Staubli VAL3: PlasticMain.pjx

--- PlasticMain.pjx ---
Parameters version=s7.0 stackSize=400000 millimeterUnit=true
Program file=__ts_english.pgx
Program file=__ts_german.pgx
Program file=__ts_swedish.pgx
Program file=_globals.pgx
Program file=changeLog.pgx
Program file=checkRobotPos.pgx
Program file=checkTaskStates.pgx
Program file=cleanUpDataBase.pgx
Program file=controlTasks.pgx
Program file=createLicense.pgx
Program file=detailedStack.pgx
Program file=loadApplication.pgx
Program file=loadLibraries.pgx
Program file=loadSysData.pgx
Program file=loadUserProgram.pgx
Program file=loadVersionInfo.pgx
Program file=logo.pgx
Program file=parseStackInfo.pgx
Program file=processEvents.pgx
Program file=run.pgx
Program file=saveApplication.pgx
Program file=start.pgx
Program file=startUpTask.pgx
Program file=status.pgx
Program file=stop.pgx
Program file=taskKill.pgx
Program file=taskKiller.pgx
Data file=PlasticMain.dtx
Library alias=rob path=Disk://Plastic/Prototypes/modRobot/modRobot.pjx autoload=false
Library alias=data path=Disk://Plastic/templates/sysDataTemplate/sysDataTemplate.pjx autoload=false
Library alias=secu path=Disk://Plastic/Prototypes/modSafety/modSafety.pjx autoload=false
Library alias=util path=Disk://Plastic/Prototypes/modBackup/modBackup.pjx autoload=false
Library alias=FUN path=Disk://Plastic/templates/tempSysFuncCall/tempSysFuncCall.pjx autoload=false
Library alias=fun path=Disk://Plastic/Prototypes/modFunction/modFunction.pjx autoload=false
Library alias=ui path=Disk://Plastic/Prototypes/modUserDisp/modUserDisp.pjx autoload=false
Library alias=prg path=Disk://Plastic/templates/tempUserProgram/tempUserProgram.pjx autoload=false
Library alias=USER path=Disk://Plastic/templates/tempIoUser/tempIoUser.pjx autoload=false
Library alias=app path=Disk://Plastic/templates/tempApplication/tempApplication.pjx
Library alias=appTmp path=Disk://Plastic/templates/tempApplication/tempApplication.pjx
Library alias=evt path=Disk://Plastic/Prototypes/modEvents/modEvents.pjx autoload=false
Library alias=SYS path=Disk://io_System/io_System.pjx
Library alias=str path=Disk://Libraries/stringHandling/stringHandling.pjx
Library alias=list path=Disk://Libraries/listHandling/listHandling.pjx
Library alias=upd path=Disk://Plastic/Prototypes/modUpdater/modUpdater.pjx autoload=false
Library alias=stat path=Disk://Plastic/Prototypes/modStatus/modStatus.pjx autoload=false
Library alias=lang path=Disk://Plastic/i18n/i18n.pjx
Library alias=db path=Disk://Plastic/Prototypes/modDatabase/modDatabase.pjx autoload=false
Library alias=usr path=Disk://Plastic/Prototypes/modUserIO/modUserIO.pjx autoload=false
Library alias=hw path=Disk://Libraries/hardware/hardware.pjx
Library alias=msl path=Disk://Plastic/Prototypes/modMsl/modMsl.pjx autoload=false
Library alias=customModule path=Disk://Plastic/Prototypes/modCustom/modCustom.pjx autoload=false
Library alias=userIO path=Disk://zUserIODef/zUserIODef.pjx autoload=false
Library alias=monitor path=Disk://Plastic/Prototypes/modMonitor/modMonitor.pjx autoload=false
Library alias=debug path=Disk://Libraries/debug/debug.pjx

--- start.pgx ---
public program start()
  local bool bResult
  local bool bLicense
begin
    //
  //\var bResult
  //\var bLicense
  //
//===========================================================================
  //   START UP ROBOT
  //===========================================================================
  cls()
  delay(0)
  userPage()
  call logo()
  call debug:setVerbosity(libPath(),debug:LEV_INFO)
  title(sCopyRight+sVersion)
  // Initialize System IO
  call SYS:InitSysIO()
  taskCreate "starting",10,startUpTask()
  // load version information
  call loadVersionInfo()
  logMsg(sCopyRight+sVersion)
  // detect hardware
  call hw:start()
  //!issue 23
  // check if a new version was installed and check dependcies of sys data library
  bResult=true
  homeFlag=false
  bFirstLoad=true
  nPLCRestartCnt=0
  // check if running on emulator
  SYS:bIsEmulator=getVersion("Starc")==""

  call loadSysData(bResult, bLicense)
  if bResult
    if bLicense
      call createLicense()
    endIf
    call loadLibraries(bResult)


    // if dependencies are ok we can proceed to start up
    //if upd:sResult==""
    if bResult
      call util:start()
      call FUN:start()
      call FUN:loadSysData("zData",bResult)
      call fun:start()
      call fun:loadSysData("zData",bResult)
      call rob:loadSysData("zData",bResult)
      call secu:loadSysData("zData",bResult)
      //    call scr_:loadSysData("zData",bResult)
      call ui:loadSysData("zData",bResult)
      delay(2)
      //!issue 22: load user program events
      call loadUserProgram(bResult)
      //
      bStartUp=false
      wait(taskStatus("starting")==-1)
      if bResult
        // initialize language
        call lang:start()
        if data:sLanguage==""
          data:sLanguage="english"
          call lang:setLanguage(data:sLanguage)
        else
          call lang:setLanguage(data:sLanguage)
        endIf

        // START UP USER DISPLAY =========================
        call ui:start()
        if ui:bStartUp
          // initialize database
          call db:start()
          //
          // Start up master/slave com
          call msl:start()
          // Start up robot
          call rob:start()

          // start IO monitor if io:monitor is defined
          call monitor:start()
          // pass on version information to UI
          ui:sVersion=sVersion
          // initiate full home return on start up
          SYS:bTotalHome=true
          //!change 16.10.06, vdg: Force a home return even if robot is already at home
          SYS:bForceHomeReq=data:setForceHome
          //
          //
          // Initialize User IO
          call USER:InitUserIO()
          // initialize custom modules
          call customModule:start()
          call run()
          // start main loop
          //taskCreate "Run",10,run()
          //call ui:popUp("Application started",data:nMsgTimeOut,false)
          //taskCreateSync "status",16,overrun,status()
        endIf
      endIf
    endIf
  endIf
  //wait(taskStatus("Run")==-1)
end

--- __ts_english.pgx ---
program __ts_english()
begin
  //
end

--- __ts_swedish.pgx ---
program __ts_swedish()
begin
  //
end

--- createLicense.pgx ---
program createLicense()
  local string txt[6]
  local string orderNumber
  local num i
 begin
    //\brief
  // Create a license key for the robot system. License key information is saved
  // in system data library
  //
  //\var txt
  //\var orderNumber
  //\var i
  //
//!brief
  // Create a license key for the robot system. License key information is saved
  // in system data library
  //
  orderNumber=getVersion("serialNumber")
  txt=""
  //!issue 36
  if data:libLoad("zData")==0
    call list:resizeNum(data:nLic,len(orderNumber))
    data:sMachineNumber=orderNumber
    for i=0 to size(data:nLic)-1
      data:nLic[i]=asc(orderNumber,i)*(i+1)
      txt=txt+toString("",asc(orderNumber,i)*(i+1))+", "
    endFor
    call data:saveData()
    popUpMsg(txt)
  else
    popUpMsg("Loading the data library failed!")
  endIf
end

--- crypt.pgx ---
program crypt()
begin
end

--- detailedStack.pgx ---
program detailedStack()
  local num i
  local num nTaskStatus
  local num count
  local num j
  local string stack[20]
begin
    //\brief
  //Write detailed stack info to log
  //\var i
  //\var nTaskStatus
  //\var count
  //\var j
  //\var stack
  //
//!brief
  //Write detailed stack info to log
  for i=0 to size(sTaskName)-1
    logMsg("Stack Information for task: "+sTaskName[i])
    nTaskStatus=taskStatus(sTaskName[i])
    // suspend the task
    if nTaskStatus==1
      taskSuspend(sTaskName[i])
    endIf
    // wait until task stopped
    wait(taskStatus(sTaskName[i])!=1)
    // retrieve call stack
    count=$taskCallStack(sTaskName[i],stack)
    // write call stack to log
    for j=0 to count-1
      logMsg(stack[j])
    endFor
    // resume task if it was active when entering this routine
    if nTaskStatus==1
      taskResume(sTaskName[i],0)
    endIf
  endFor
end

--- loadApplication.pgx ---
program loadApplication(string name_)
  local num nResult
  local string txt[4]
begin
    //\brief
  //
  //\fix
  //03.05.06, vdg: Halt all tasks while loading the new application
  // This should avoid "pure virtual function calls" and "page faults"
  //\fix
  //11.03.08, vdg: Load correct template library for user application
  //\var nResult
  //\var txt
  //\param name_
  //
//!fix 03.05.06, vdg: Halt all tasks while loading the new application
  //                    This should avoid "pure virtual function calls" and "page faults"
  //!fix 11.03.08, vdg: Load correct template library for user application
  call rob:haltTasks()
  //!change 23.05.06, vdg: unload the application from application manager only if reloading the
  // same application again
  if name_==data:sApplication
    //!fixme 09.10.06, vdg: make sure that reloading the same application works
    logMsg("Closing library in app manager: "+name_)
    app:$libClose()
    logMsg("Library closed")
    delay(2)
    logMsg("Loading library alias")
    nResult=appTmp:libLoad("Plastic/templates/tempApplication")
    logMsg("return code for temp load: "+toString("",nResult))
    delay(2)
    nResult=app:libLoad("Plastic/templates/tempApplication")
    logMsg("return code: "+toString("",nResult))
    delay(2)
    logMsg("Loading alias done")
  endIf
  // try to load the application
  nResult=app:libLoad(name_)
  // check if loading was successfull
  if nResult!=0
    // inform operator what public symbos are missing in case of loading error 11 ==> interface mismatch
    if nResult==11
      if !app:libExist("HR_HomeReturn()")
        call str:printf1arg((("The routine /tiHR_HomeReturn/tn is not defined or not set public in application /ti%1/tn.")),name_,txt)
        call ui:popUp(txt,0,true)
      endIf
      if !app:libExist("MP_MainProgram()")
        call str:printf1arg((("The routine /tiMP_MainProgram/tn is not defined or not set public in application /ti%1/tn.")),name_,txt)
        call ui:popUp(txt,0,true)
      endIf
      if !app:libExist("PLC_MainPLC()")
        call str:printf1arg((("The routine /tiPLC_MainPLC/tn is not defined or not set public in application /ti%1/tn.")),name_,txt)
        call ui:popUp(txt,0,true)
      endIf
      if !app:libExist("tGripCenter")
        call str:printf1arg((("The global data /titGripCenter/tn of type tool is not defined or not set public in application /ti%1/tn.")),name_,txt)
        call ui:popUp(txt,0,true)
      endIf
      if !app:libExist("jHome")
        call str:printf1arg((("The global data /tijHome/tn of type joint is not defined or not set public in application /ti%1/tn.")),name_,txt)
        call ui:popUp(txt,0,true)
      endIf
    endIf
    // revert changes and reload the old application
    //!change 05.04.06, vdg: add information to log
    call str:printf3arg((("Loading application %1 failed: %2 %3")),name_,toString("0.0",nResult),ui:sLibraryMessage[min(nResult,size(ui:sLibraryMessage)-1)],txt)
    call ui:popUp(txt,0,true)
    logMsg(txt)
    //!change 06.06.06, vdg: if reloading the old application also fails, reload
    //  the standard library z01_Application
    nResult=app:libLoad(data:sApplication)
    if nResult!=0
      app:libLoad("Plastic/templates/tempApplication")
      data:sApplication=""
    endIf
  else
    //!Issue 22: call user event program
    call prg:onAppLoad(name_)
    //!change 05.04.06, vdg: add information to log
    logMsg("Application "+name_+" loaded")
    //!change 23.05.06, vdg: load application in application manager
    //!fixme 07.08.06, vdg: sometimes loading a library with $libOpen crashes the application manager
    // thus $libOpen() removed again.
    app:$libOpen()
    //delay(5)
    data:sApplication=name_
    //!todo 03.05.06, vdg: For some reason saving data causes a page fault here
    //data:libSave()
    //!issue 42: reset auxilary buttons
    SYS:sAux1=""
    SYS:sAux2=""
    SYS:nLiAux1=0
    SYS:nLiAux2=0
  endIf
  SYS:bFirstRunAfterL=true
  SYS:bModified=false
  data:jHome=app:jHome
  //!fix 10.05.06, vdg: do not copy the entire structure as this will create undefined references
  //                    when app is being replaced by a libLoad() instruction
  data:tTCP.trsf=app:tGripCenter.trsf
  //!fix 05.04.06, vdg: relink IO to make them effective in application... is this a bug?
  call usr:clearUserIO()
  call usr:clearUserMon()
  //!fix 22.05.06, vdg: reset gripper links if user gripper signals are used
  //if !data:setSystemGrip
  //call ui:clearGripperIO()
  //endIf
  call SYS:InitSysIO()
  call USER:InitUserIO()
  //!fix 03.05.06, vdg: restart all tasks
  call rob:restart()
  data:libSave()
end

--- loadSysData.pgx ---
program loadSysData(bool& bResult_[], bool& bSetupLicense_[])
  local num nResult
begin
    //
  //\var nResult
  //\param bResult_
  //\param bSetupLicense_
  //
put("Loading Data for: "+libPath()+" :")
  nResult=data:libLoad("zData")
  bSetupLicense_=false
  //
  switch true
    // library loaded
    case nResult==0
      putln("ok")

    break
    // zData library does not exist yet, so we save the template
    // as zData
    case nResult>=30
      bResult_=false
      logMsg("zData not found!")
      // reload template
      nResult=data:libLoad("Plastic/templates/sysDataTemplate")
      if nResult==0
        // save template as zData
        nResult=data:libSave("zData")
        if nResult==0
          logMsg("zData recreated from template")
          bResult_=true
          // if profile 'swiss-system' is active also force creation of license
          if getProfile()=="swiss-system"
            bSetupLicense_=true
          else
            popUpMsg("A new zData library has been created. Please reinstall runtime license!")
          endIf
        else
          logMsg("Creating zData failed!")
        endIf
      endIf
    break
    // library load failed for some other reason
    default
      putln("failed")
      putln("Checking data dependencies")
      call upd:checkDepend()
      bResult_=false
    break
  endSwitch
end

--- loadVersionInfo.pgx ---
program loadVersionInfo()
  local num handle
begin
    //\brief
  //Load version information and build information from external file.
  //
  //The file Disk://Plastic/version.dat is loaded and the first line is used as version number.
  //The file Disk://Plastic/build.dat is loaded and the first line is used as build number.
  //\var handle
  //
//!brief
  //Load version information and build information from external file.
  //
  //The file Disk://Plastic/version.dat is loaded and the first line is used as version number.
  //The file Disk://Plastic/build.dat is loaded and the first line is used as build number.
  sVersion="unknown"
  handle=$fileOpen("Disk://Plastic/version.dat","r")
  if handle>=0
    $fileGet(handle,sVersion,1)
    $fileClose(handle)
  endIf
  sBuildNumber="unknown"
  handle=$fileOpen("Disk://Plastic/build.dat","r")
  if handle>=0
    $fileGet(handle,sBuildNumber,1)
    $fileClose(handle)
  endIf
  logMsg("Build: "+sBuildNumber)
end

--- parseStackInfo.pgx ---
program parseStackInfo(string stackInfo_, string& library_[], string& program_[], num& line_[], string& code_[])
  local bool error
  local string dummy
begin
    //
  //\var error
  //\var dummy
  //\param stackInfo_
  //\param library_
  //\param program_
  //\param line_
  //\param code_
  //
if len(stackInfo_)>0
    library_=left(stackInfo_,find(stackInfo_,":"))
    stackInfo_=right(stackInfo_,len(stackInfo_)-find(stackInfo_,":")-1)
    program_=left(stackInfo_,find(stackInfo_,")")+1)
    stackInfo_=right(stackInfo_,len(stackInfo_)-find(stackInfo_,")")-1)
    stackInfo_=right(stackInfo_,len(stackInfo_)-find(stackInfo_,"ne")-3)
    dummy=stackInfo_
    dummy=toNum(dummy,line_,error)
    stackInfo_=right(stackInfo_,len(stackInfo_)-find(stackInfo_,":")-1)
    code_=stackInfo_
  endIf
end

--- run.pgx ---
program run()
  local num idx
begin
    //\brief
  //
  //\change
  //27.04.6, vdg: Added information if home return is active (SYS:bHomeRetActive)
  //\change
  //23.04.06, vdg: - clear all pending status messages that are not persistent
  // - reset pallet counters after a total home return
  //\change
  //07.06.06, vdg: - code clean up: move code to sub routines
  //
  //\var idx
  //
//!change 27.04.6, vdg: Added information if home return is active (SYS:bHomeRetActive)
  //!change 23.04.06, vdg: - clear all pending status messages that are not persistent
  //                       - reset pallet counters after a total home return
  //!change 07.06.06, vdg: - code clean up: move code to sub routines
  //
  for idx=0 to size(stat:nTaskState)-1
    stat:nTaskState[idx]=-1
  endFor
  //
  //!Issue 22: call user event program
  call prg:onSystemStart()
  call prg:startPLC()
  while (rob:bRobActive)
    delay(0)
    call processEvents()
    call checkRobotPos()
    call checkTaskStates(stat:nTaskState)
    call controlTasks()
    // run rob module synchronously
    if !data:setAsyncRun
      call rob:run()
    endIf
  endWhile
  call prg:stopPLC()
end

--- saveApplication.pgx ---
program saveApplication()
  local num nResult
begin
    //
  //\var nResult
  //
// save the application
  nResult=app:libSave()
  // check if saving was successfull
  if nResult!=0
    popUpMsg("Saving Application failed: "+toString("",nResult))
  else
    SYS:bModified=false
  endIf
  data:libSave()
end

--- status.pgx ---
program status()
  local num count
  local string callStack
  local string library
  local string program
  local num line
  local string code
begin
    //
  //\var count
  //\var callStack
  //\var library
  //\var program
  //\var line
  //\var code
  //
while true
    count=$taskCallStack(sTaskName[1],callStack)
    call parseStackInfo(callStack,library,program,line,code)
    if program=="SP_Traj"
      call list:resizeString(programList,max(size(programList),line))
      programList[line]=code
    endIf
  endWhile
end

--- taskKill.pgx ---
program taskKill(string sTaskName_, bool& bResult_[])
  local num idx
begin
    //\brief
  //The program tries to kill task sTaskName_. bResult_ is false if it does not
  // succeed within 2 sec
  //\var idx
  //\param sTaskName_ The name of the task that should be killed
  //\param bResult_ The result of the kill operation
  //
  // find free task
  //
//!brief
  //The program tries to kill task sTaskName_. bResult_ is false if it does not
  // succeed within 2 sec
  //!param sTaskName_ : The name of the task that should be killed
  //!param bResult_   : The result of the kill operation
  //
  // find free task
  idx=0
  while taskStatus("killer"+toString("",idx))!=-1
    idx=idx+1
  endWhile
  taskCreate "killer"+toString("",idx),1,taskKiller(sTaskName_)
  if !watch(taskStatus("killer"+toString("",idx))==-1,2)
    bResult_=false
    taskKill("killer"+toString("",idx))
  else
    bResult_=true
  endIf
end

--- taskKiller.pgx ---
program taskKiller(string sTask_)
begin
    //
  //\param sTask_
  //
taskKill(sTask_)
end
